// TIA Portal V17 export
// export: Created 2022-07-20T07:01:27.512878Z, ExportSetting WithDefaults, DisplayName Totally Integrated Automation Portal, DisplayVersion V17, DisplayName TIA Portal Openness, DisplayVersion V17, DisplayName TIA Portal Version Control Interface, DisplayVersion V17, DisplayName SINAMICS Startdrive Advanced, DisplayVersion V17, DisplayName SINAMICS Startdrive G130, G150, S120, S150, SINAMICS MV, S210, DisplayVersion V17, DisplayName SINAMICS Startdrive G110M, G120, G120C, G120D, G120P, G115D, DisplayVersion V17, DisplayName STEP 7 Professional, DisplayVersion V17, DisplayName STEP 7 Safety, DisplayVersion V17, DisplayName WinCC Advanced, DisplayVersion V17
FUNCTION_BLOCK "FB10271_HiwinAlphajetDoor"   // FB10271, LAD
{ S7_Optimized_Access := 'TRUE' }
VERSION : 0.1
// You can manage the maximum time for opening with the variable "Max_Time_OpenClose"
// stored: AutoNumber false, IsIECCheckEnabled false, IsRetainMemResEnabled false, MemoryReserve 100, SetENOAutomatically false, UDAEnableTagReadback false
   VAR_INPUT
      Opening_Authorization : Bool;
      PushButton : Bool;
      Door_Sensor : Bool;
      Clock_light : Bool;
   END_VAR
   VAR_OUTPUT
      Door_Closed : Bool;
   END_VAR
   VAR_IN_OUT
      Led_PushButton : Bool;
      Out_Actuator_Activation : Bool := false;
      Out_Actuator_Direction : Bool := false;
   END_VAR
   VAR
      Long_Press : Bool;
      Short_Press : Bool;
      OnLongPress { S7_SetPoint := 'True'} : Bool;
      Door_Opened : Bool;
      Time_Used_For_Opening : Time;
      Time_Used_For_Closing : Time := T#0MS;
      Time_Remaining : Time := T#10s;
      Calc_Time_Remaining : Bool;
      Put_Result : Bool;
      Enable_Actuator : Bool := false;
      Disable_Actuator : Bool;
      Reset_Timer_Door_Closing { ExternalAccessible := 'False'; ExternalVisible := 'False'; ExternalWritable := 'False'} : Bool;
      Result_Calc_TIme_Remaining : Time;
      Reset_Timer_Door_Opening : Bool;
      Rising_ShortPress : Bool;
      Falling_OnLongPress : Bool;
      Max_Time_OpenClose { S7_SetPoint := 'True'} : Time := T#10s;
      FB_Detect_PushType_Instance { S7_SetPoint := 'True'} : "FB10040_Button_DetectPushType";
      TON_Enable_Actuator_Activation { S7_SetPoint := 'True'} : TON_TIME;
      TP_Enable_Actuator_Activation { S7_SetPoint := 'True'} : TP_TIME;
      TP_Disable_Actuator { S7_SetPoint := 'True'} : TP_TIME;
      TONR_Door_Closing { S7_SetPoint := 'True'} : TONR_TIME;
      TONR_Door_Opening { S7_SetPoint := 'True'} : TONR_TIME;
      TON_Time_Before_Stop { S7_SetPoint := 'True'} : TON_TIME;
      R_TRIG_Door_Sensor : R_TRIG;
   END_VAR
   VAR_TEMP   // added for the SCL form of the ladder/FBD networks
      _w1 : Bool;
      _w2 : Bool;
   END_VAR
BEGIN

REGION Network 1: Detect Short/Long Press
   // Detect Short / Long Press
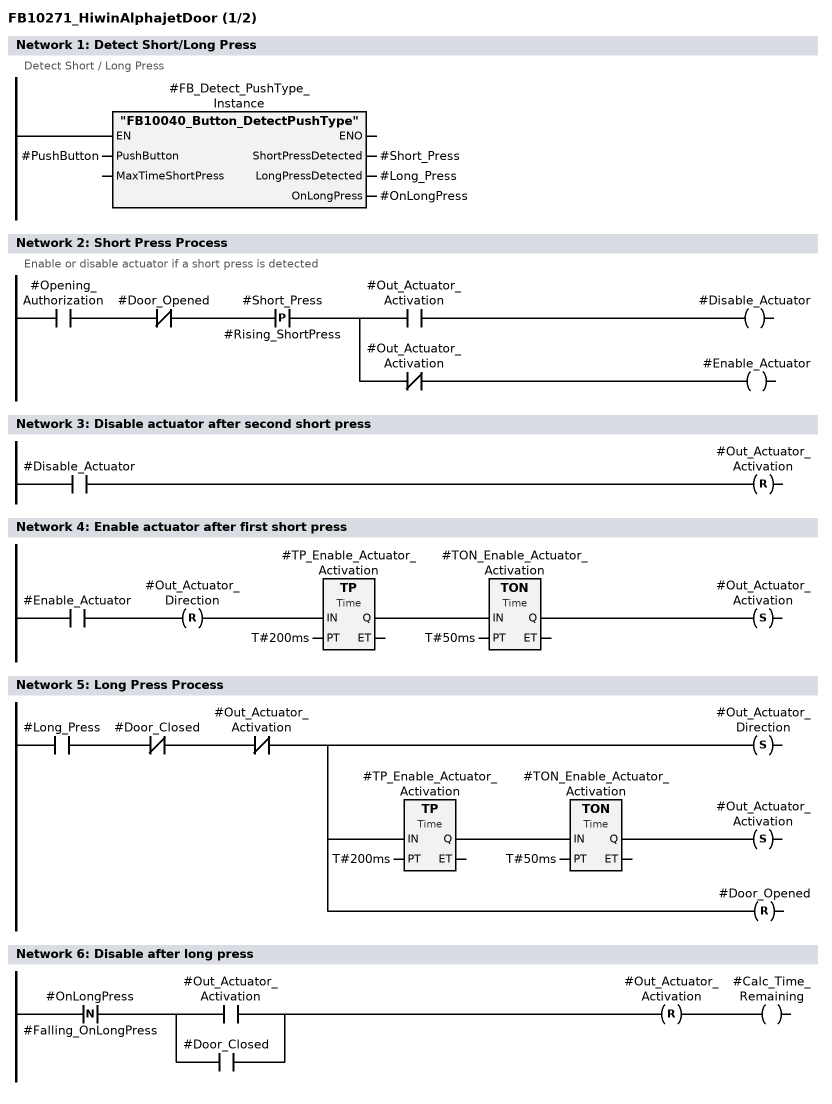
   RUNG wire#powerrail
      #FB_Detect_PushType_Instance(PushButton := #PushButton, MaxTimeShortPress :=, ShortPressDetected => #Short_Press, LongPressDetected => #Long_Press, OnLongPress => #OnLongPress)
   END_RUNG
   // the same network as SCL:
   #FB_Detect_PushType_Instance(PushButton := #PushButton,   // "FB10040_Button_DetectPushType"
                           ShortPressDetected => #Short_Press,
                           LongPressDetected => #Long_Press,
                           OnLongPress => #OnLongPress);
END_REGION

REGION Network 2: Short Press Process
   // Enable or disable actuator if a short press is detected
   RUNG wire#powerrail
      Contact( #Opening_Authorization )
      I_Contact( #Door_Opened )
      P_Contact(operand := #Short_Press, bit := #Rising_ShortPress)
      wire#w1
      Contact( #Out_Actuator_Activation )
      Coil( #Disable_Actuator )
   END_RUNG
   RUNG wire#w1
      I_Contact( #Out_Actuator_Activation )
      Coil( #Enable_Actuator )
   END_RUNG
   // the same network as SCL:
   #_w1 := #Opening_Authorization AND NOT #Door_Opened AND #Short_Press AND NOT #Rising_ShortPress;   // rising edge of #Short_Press
   #Rising_ShortPress := #Short_Press;
   #Disable_Actuator := #_w1 AND #Out_Actuator_Activation;
   #Enable_Actuator := #_w1 AND NOT #Out_Actuator_Activation;
END_REGION

REGION Network 3: Disable actuator after second short press
   RUNG wire#powerrail
      Contact( #Disable_Actuator )
      R_Coil( #Out_Actuator_Activation )
   END_RUNG
   // the same network as SCL:
   IF #Disable_Actuator THEN #Out_Actuator_Activation := FALSE; END_IF;
END_REGION

REGION Network 4: Enable actuator after first short press
   RUNG wire#powerrail
      Contact( #Enable_Actuator )
      R_Coil( #Out_Actuator_Direction )
      { S7_Templates := "time_type := Time" } #TP_Enable_Actuator_Activation.TP(pt := T#200ms, et =>)
      { S7_Templates := "time_type := Time" } #TON_Enable_Actuator_Activation.TON(pt := T#50ms, et =>)
      S_Coil( #Out_Actuator_Activation )
   END_RUNG
   // the same network as SCL:
   IF #Enable_Actuator THEN #Out_Actuator_Direction := FALSE; END_IF;
   #TP_Enable_Actuator_Activation(IN := #Enable_Actuator, PT := T#200ms);   // TP
   #TON_Enable_Actuator_Activation(IN := #TP_Enable_Actuator_Activation.Q, PT := T#50ms);   // TON
   IF #TON_Enable_Actuator_Activation.Q THEN #Out_Actuator_Activation := TRUE; END_IF;
END_REGION

REGION Network 5: Long Press Process
   RUNG wire#powerrail
      Contact( #Long_Press )
      I_Contact( #Door_Closed )
      I_Contact( #Out_Actuator_Activation )
      wire#w1
      S_Coil( #Out_Actuator_Direction )
   END_RUNG
   RUNG wire#w1
      { S7_Templates := "time_type := Time" } #TP_Enable_Actuator_Activation.TP(pt := T#200ms, et =>)
      { S7_Templates := "time_type := Time" } #TON_Enable_Actuator_Activation.TON(pt := T#50ms, et =>)
      S_Coil( #Out_Actuator_Activation )
   END_RUNG
   RUNG wire#w1
      R_Coil( #Door_Opened )
   END_RUNG
   // the same network as SCL:
   #_w1 := #Long_Press AND NOT #Door_Closed AND NOT #Out_Actuator_Activation;
   IF #_w1 THEN #Out_Actuator_Direction := TRUE; END_IF;
   #TP_Enable_Actuator_Activation(IN := #_w1, PT := T#200ms);   // TP
   #TON_Enable_Actuator_Activation(IN := #TP_Enable_Actuator_Activation.Q, PT := T#50ms);   // TON
   IF #TON_Enable_Actuator_Activation.Q THEN #Out_Actuator_Activation := TRUE; END_IF;
   IF #_w1 THEN #Door_Opened := FALSE; END_IF;
END_REGION

REGION Network 6: Disable after long press
   RUNG wire#powerrail
      N_Contact(operand := #OnLongPress, bit := #Falling_OnLongPress)
      wire#w1
      Contact( #Out_Actuator_Activation )
      wire#w2
      R_Coil( #Out_Actuator_Activation )
      Coil( #Calc_Time_Remaining )
   END_RUNG
   RUNG wire#w1
      Contact( #Door_Closed )
   END_RUNG wire#w2
   // the same network as SCL:
   #_w1 := NOT #OnLongPress AND #Falling_OnLongPress;   // falling edge of #OnLongPress
   #Falling_OnLongPress := #OnLongPress;
   #_w2 := #_w1 AND (#Out_Actuator_Activation OR #Door_Closed);
   IF #_w2 THEN #Out_Actuator_Activation := FALSE; END_IF;
   #Calc_Time_Remaining := #_w2;
END_REGION

REGION Network 7 (SCL): Check if door closed
   // The remaining time > max time  is not necessary
   IF (#Time_Remaining > #Max_Time_OpenClose) OR #R_TRIG_Door_Sensor.Q  THEN
       #Time_Remaining := #Max_Time_OpenClose;
       #Put_Result := TRUE;
       #Put_Result := FALSE;
   END_IF;
END_REGION

REGION Network 8 (SCL): Stop if door closed
   // If the door is closed and the requested instruction is closing, the instruction is stopped.
   IF (#Out_Actuator_Activation AND #Out_Actuator_Direction AND #Door_Sensor) OR #Door_Opened THEN
       #Out_Actuator_Direction := FALSE;
       #Out_Actuator_Activation := FALSE;

   END_IF;
END_REGION

REGION Network 9 (SCL): LED & Door Sensor
   // Turn on the light to indicate that the door can be used     |     The information on the door status   |    Flashes the led if the door is not closed and there is no authorization
   #Door_Closed := #Door_Sensor;

   IF #Opening_Authorization THEN
       #Led_PushButton := TRUE;
   ELSE
       IF NOT #Door_Closed AND NOT #Opening_Authorization THEN
           #Led_PushButton := #Clock_light;
       ELSE
           #Led_PushButton := FALSE;
       END_IF;

   END_IF;
END_REGION

REGION Network 10 (SCL): Calculation Time Remaining
   // Add or subtract time from the remaining time if the door opens or closes
   IF  (#Calc_Time_Remaining OR #Disable_Actuator) AND NOT #Put_Result THEN
       IF NOT #Out_Actuator_Direction THEN
           #Result_Calc_TIme_Remaining := #Time_Remaining - #Time_Used_For_Opening;
           #Reset_Timer_Door_Opening := TRUE;
       ELSE
           #Result_Calc_TIme_Remaining := #Time_Remaining + #Time_Used_For_Closing;
           #Reset_Timer_Door_Closing := TRUE;
       END_IF;
       #Put_Result := TRUE;
   END_IF;
END_REGION

REGION Network 11 (SCL): Put Result
   IF #Put_Result THEN
       #Time_Remaining := #Result_Calc_TIme_Remaining;
       #Put_Result := FALSE;
   END_IF;
END_REGION

REGION Network 12: Check time used for opening
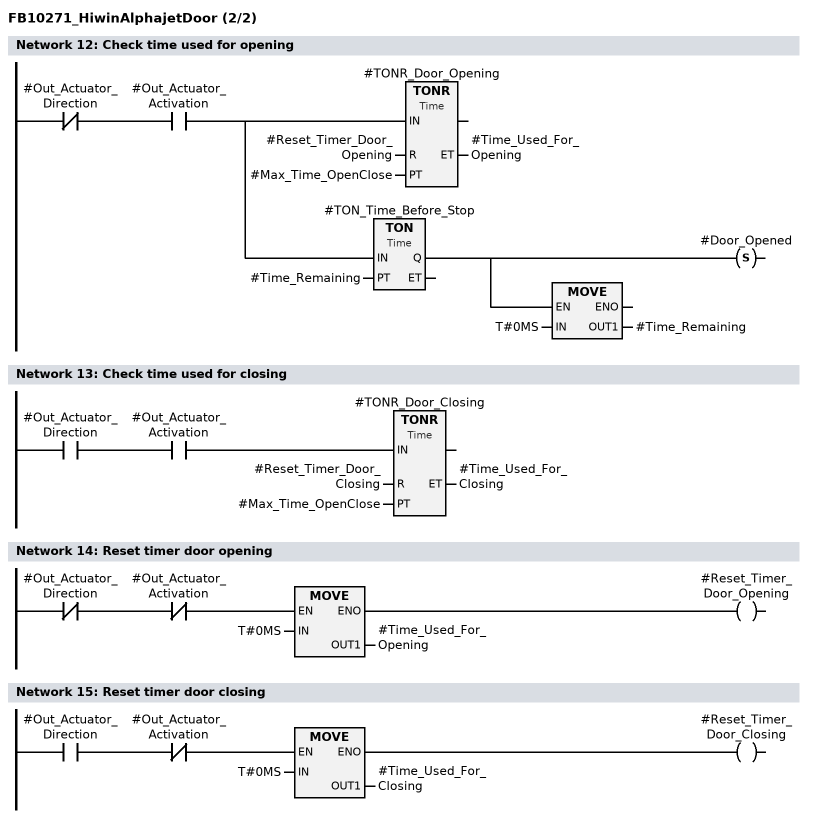
   RUNG wire#powerrail
      I_Contact( #Out_Actuator_Direction )
      Contact( #Out_Actuator_Activation )
      wire#w1
      { S7_Templates := "time_type := Time" } #TONR_Door_Opening.TONR(r := #Reset_Timer_Door_Opening, pt := #Max_Time_OpenClose, et => #Time_Used_For_Opening)
   END_RUNG
   RUNG wire#w1
      { S7_Templates := "time_type := Time" } #TON_Time_Before_Stop.TON(pt := #Time_Remaining, et =>)
      wire#w2
      S_Coil( #Door_Opened )
   END_RUNG
   RUNG wire#w2
      Move(in := T#0MS, out1 => #Time_Remaining)
   END_RUNG
   // the same network as SCL:
   #_w1 := NOT #Out_Actuator_Direction AND #Out_Actuator_Activation;
   #TONR_Door_Opening(IN := #_w1,   // TONR
                      R := #Reset_Timer_Door_Opening,
                      PT := #Max_Time_OpenClose,
                      ET => #Time_Used_For_Opening);
   #TON_Time_Before_Stop(IN := #_w1, PT := #Time_Remaining);   // TON
   IF #TON_Time_Before_Stop.Q THEN
       #Door_Opened := TRUE;
       #Time_Remaining := T#0MS;
   END_IF;
END_REGION

REGION Network 13: Check time used for closing
   RUNG wire#powerrail
      Contact( #Out_Actuator_Direction )
      Contact( #Out_Actuator_Activation )
      { S7_Templates := "time_type := Time" } #TONR_Door_Closing.TONR(r := #Reset_Timer_Door_Closing, pt := #Max_Time_OpenClose, et => #Time_Used_For_Closing)
   END_RUNG
   // the same network as SCL:
   #TONR_Door_Closing(IN := #Out_Actuator_Direction AND #Out_Actuator_Activation,   // TONR
                      R := #Reset_Timer_Door_Closing,
                      PT := #Max_Time_OpenClose,
                      ET => #Time_Used_For_Closing);
END_REGION

REGION Network 14: Reset timer door opening
   RUNG wire#powerrail
      I_Contact( #Out_Actuator_Direction )
      I_Contact( #Out_Actuator_Activation )
      Move(in := T#0MS, out1 => #Time_Used_For_Opening)
      Coil( #Reset_Timer_Door_Opening )
   END_RUNG
   // the same network as SCL:
   #_w1 := NOT #Out_Actuator_Direction AND NOT #Out_Actuator_Activation;
   IF #_w1 THEN #Time_Used_For_Opening := T#0MS; END_IF;
   #Reset_Timer_Door_Opening := #_w1;
END_REGION

REGION Network 15: Reset timer door closing
   RUNG wire#powerrail
      Contact( #Out_Actuator_Direction )
      I_Contact( #Out_Actuator_Activation )
      Move(in := T#0MS, out1 => #Time_Used_For_Closing)
      Coil( #Reset_Timer_Door_Closing )
   END_RUNG
   // the same network as SCL:
   #_w1 := #Out_Actuator_Direction AND NOT #Out_Actuator_Activation;
   IF #_w1 THEN #Time_Used_For_Closing := T#0MS; END_IF;
   #Reset_Timer_Door_Closing := #_w1;
END_REGION

REGION Network 16 (SCL): Edge Signals
   REGION EDGE SIGNALS
       #R_TRIG_Door_Sensor(CLK := #Door_Sensor);
   END_REGION
END_REGION
END_FUNCTION_BLOCK
